VAR_GLOBAL

// VGC Valves

{attribute 'pytmc' := ' pv: fb_TV1K0_GAS_VGC_1 '}
fb_TV1K0_GAS_VGC_1 : FB_VGC;

END_VAR

(* stored: Version 1.1.0.1, ProductVersion 3.1.4022.12
   GVL GVL_TV1K0_GAS_VGC_1: Id {404621a7-706f-4b2e-87bf-c7769828fd28} *)
